PROGRAM MAIN
VAR
	//fbTof : TOF := (PT := T#10S);
	fbTrig : R_TRIG;
	bBool : BOOL;
	trigCounter : ULINT;
END_VAR

//fbTof(IN := bBool);
fbTrig(CLK := bBool);
IF fbTrig.Q THEN
	trigCounter := trigCounter + 1;
END_IF

END_PROGRAM

(* stored: Version 1.1.0.1, ProductVersion 3.1.4024.12
   POU MAIN: Id {487b9517-2d2f-4621-b241-8b3ce99202ca}, SpecialFunc None *)
